(* IEC 61131-3 sources: CodesysTest/alpha/export/FBs/Cylinders/FB_ThreePositionCylinderWithFeedback.pou/Faulted.prop, 1 file *)

(* ---- Get.pm.st ---- *)
(*#-#-#-#-#-#-#-#-#-#---Declaration---#-#-#-#-#-#-#-#-#-#-#-#-#*)

VAR
END_VAR
(*#-#-#-#-#-#-#-#-#-#---Implementation---#-#-#-#-#-#-#-#-#-#-#-#-#*)

Faulted := faultIndication;
